TYPE hw_lamp_location:
    (Off_hw_lamp_location, On_hw_lamp_location);
END_TYPE

(* stored: ProductVersion 3.1.0.18, Version 1.1.0.1 *)
